// TIA Portal V17 export
// export: Created 2025-03-05T08:02:40.8398628Z, ExportSetting WithDefaults, DisplayName Totally Integrated Automation Portal, DisplayVersion V17 Update 8, DisplayName TIA Portal Openness, DisplayVersion V17 Update 8, DisplayName TIA Portal Version Control Interface, DisplayVersion V17, DisplayName SINAMICS Startdrive Advanced, DisplayVersion V17 SP2, DisplayName SINAMICS Startdrive G110M, G120, G120C, G120D, G120P, G115D, DisplayVersion V17 SP2, DisplayName SINAMICS Startdrive G130, G150, S120, S150, SINAMICS MV, S210, DisplayVersion V17 SP2, DisplayName STEP 7 Professional, DisplayVersion V17 Update 8, DisplayName SINUMERIK ONE STEP 7 Toolbox, DisplayVersion V17 Update 12, DisplayName SINUMERIK 840D sl STEP 7 Toolbox, DisplayVersion V17 Update 12, DisplayName STEP 7 Safety, DisplayVersion V17 Update 6, DisplayName WinCC Advanced, DisplayVersion V17 Update 8
FUNCTION "FC441_POWDER_FEEDERS_ALARM_DECODING" : Void   // FC441, LAD
{ S7_Optimized_Access := 'FALSE' }
AUTHOR : ETXETAR
VERSION : 1.0
// stored: AutoNumber false, IsIECCheckEnabled false, SetENOAutomatically false, UDAEnableTagReadback false
   VAR_TEMP
      RST_ALARMS_1 : Bool;   // RESET ALARMS 1
      RST_ALARMS_2 : Bool;   // RESET ALARMS 2
      ZERO : Int;   // ZERO
      RET_VAL_1 : Int;   // RET VALUE
   END_VAR
   VAR CONSTANT
      FC_CONSTANT : Int := 442;
   END_VAR
   VAR_TEMP   // added for the SCL form of the ladder/FBD networks
      _w1 : Bool;
      _w2 : Bool;
      _w3 : Bool;
   END_VAR
BEGIN

REGION Network 1: ZERO
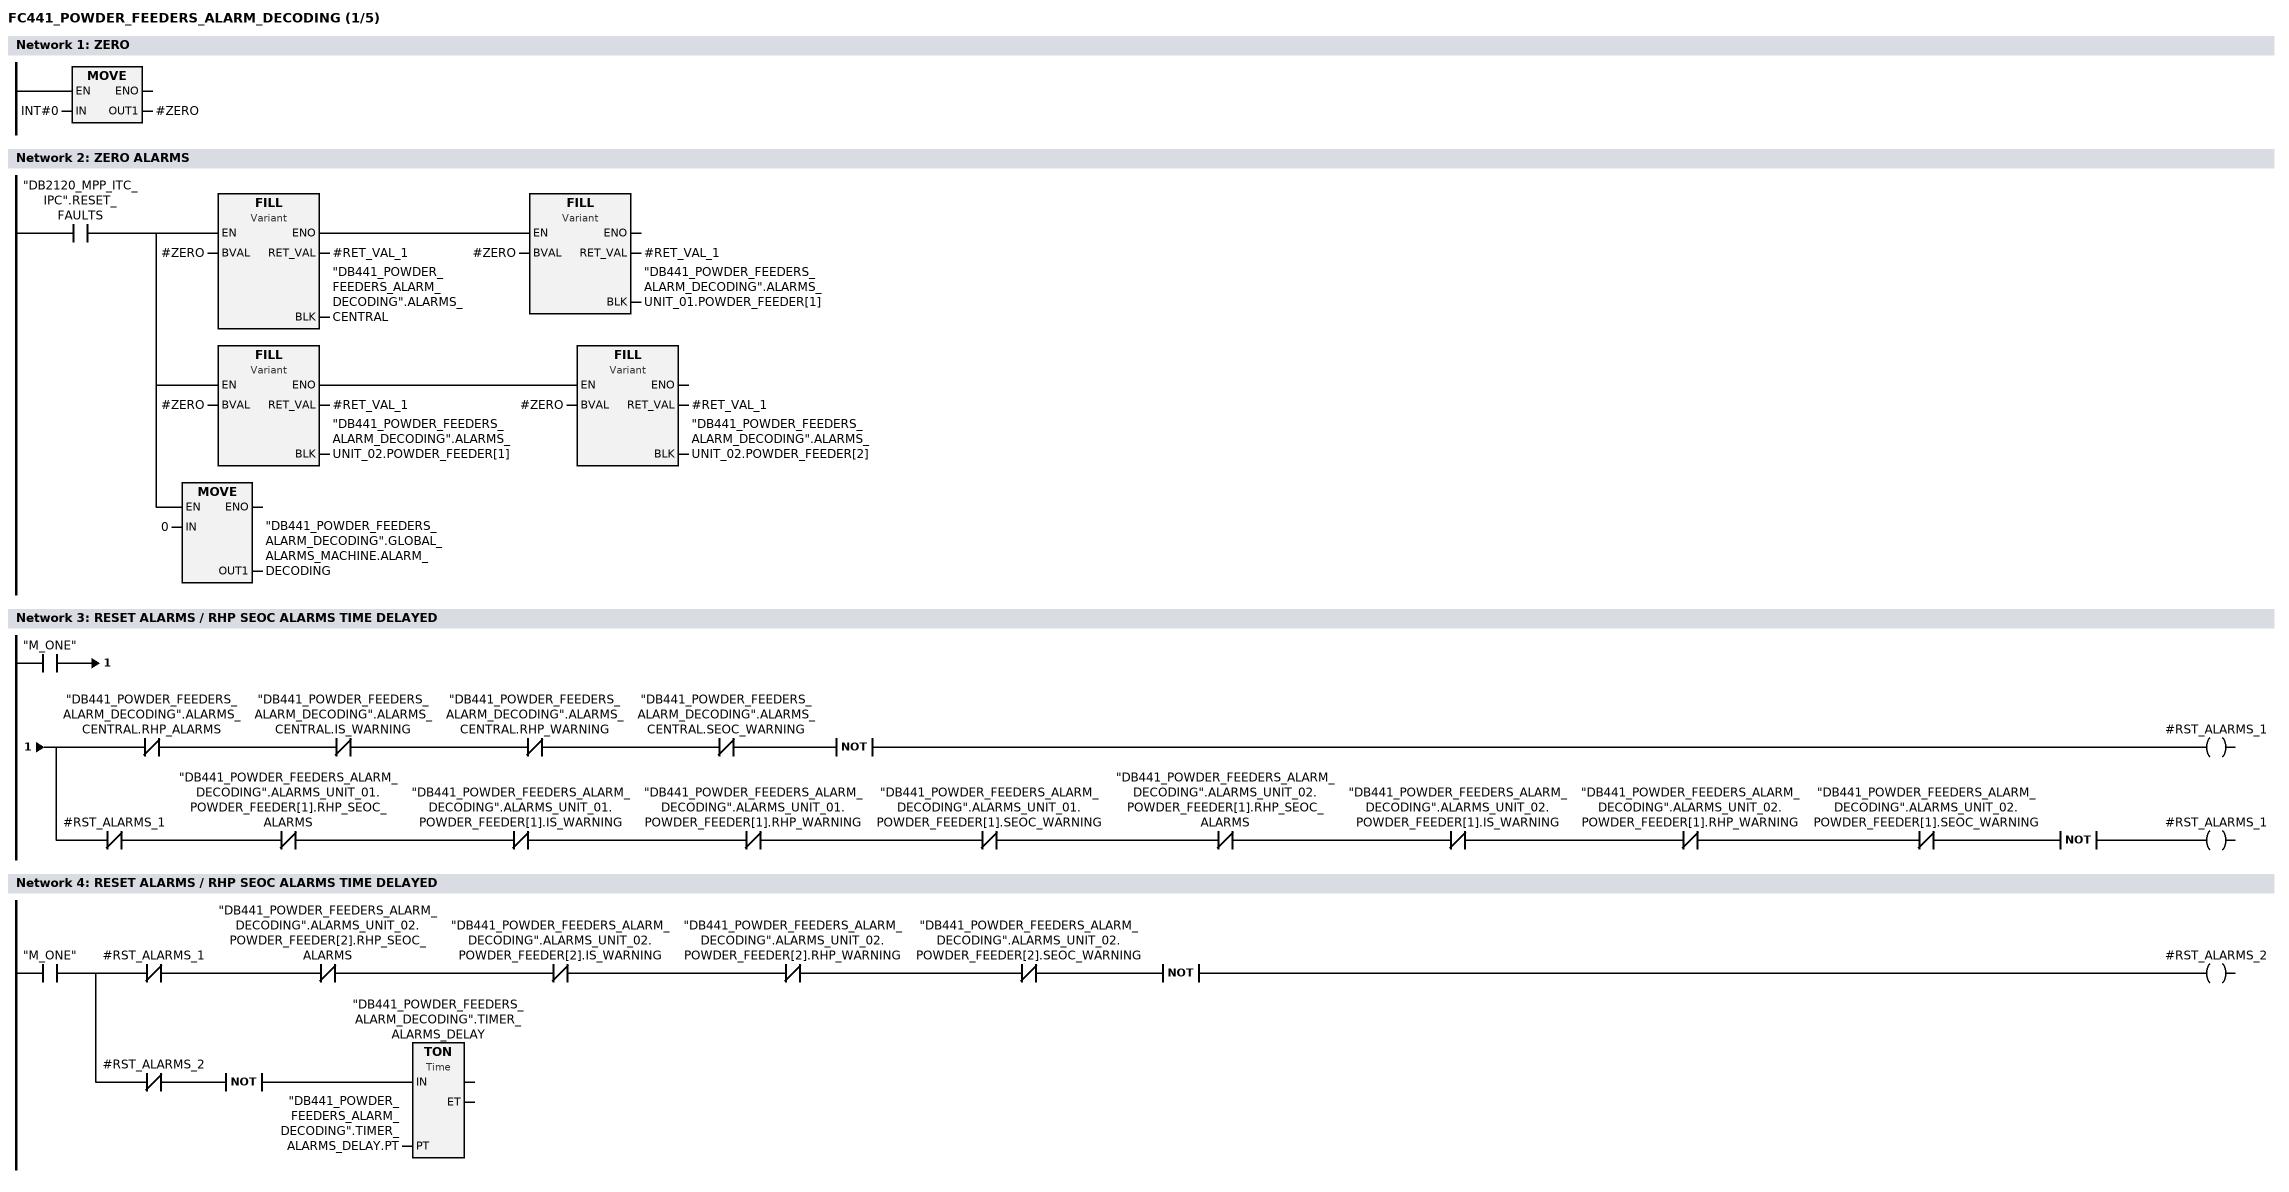
   RUNG wire#powerrail
      { S7_GenerateENO := "TRUE" } Move(in := INT#0, out1 => #ZERO)
   END_RUNG
   // the same network as SCL:
   #ZERO := INT#0;
END_REGION

REGION Network 2: ZERO ALARMS
   RUNG wire#powerrail
      Contact( "DB2120_MPP_ITC_IPC".RESET_FAULTS )
      wire#w1
      { S7_Templates := "ptr_type := Variant" } FILL(BVAL := #ZERO, RET_VAL => #RET_VAL_1, BLK => "DB441_POWDER_FEEDERS_ALARM_DECODING".ALARMS_CENTRAL)
      { S7_Templates := "ptr_type := Variant" } FILL(BVAL := #ZERO, RET_VAL => #RET_VAL_1, BLK => "DB441_POWDER_FEEDERS_ALARM_DECODING".ALARMS_UNIT_01.POWDER_FEEDER[1])
   END_RUNG
   RUNG wire#w1
      { S7_Templates := "ptr_type := Variant" } FILL(BVAL := #ZERO, RET_VAL => #RET_VAL_1, BLK => "DB441_POWDER_FEEDERS_ALARM_DECODING".ALARMS_UNIT_02.POWDER_FEEDER[1])
      { S7_Templates := "ptr_type := Variant" } FILL(BVAL := #ZERO, RET_VAL => #RET_VAL_1, BLK => "DB441_POWDER_FEEDERS_ALARM_DECODING".ALARMS_UNIT_02.POWDER_FEEDER[2])
   END_RUNG
   RUNG wire#w1
      { S7_GenerateENO := "TRUE" } Move(in := 0, out1 => "DB441_POWDER_FEEDERS_ALARM_DECODING".GLOBAL_ALARMS_MACHINE.ALARM_DECODING)
   END_RUNG
   // the same network as SCL:
   #_w2 := "DB2120_MPP_ITC_IPC".RESET_FAULTS;
   #RET_VAL_1 := FILL(EN := "DB2120_MPP_ITC_IPC".RESET_FAULTS,
                      BVAL := #ZERO,
                      BLK => "DB441_POWDER_FEEDERS_ALARM_DECODING".ALARMS_CENTRAL,
                      ENO => #_w1);
   IF #_w1 THEN
       #RET_VAL_1 := FILL(BVAL := #ZERO,
                          BLK => "DB441_POWDER_FEEDERS_ALARM_DECODING".ALARMS_UNIT_01.POWDER_FEEDER[1]);
   END_IF;
   #RET_VAL_1 := FILL(EN := #_w2,
                      BVAL := #ZERO,
                      BLK => "DB441_POWDER_FEEDERS_ALARM_DECODING".ALARMS_UNIT_02.POWDER_FEEDER[1],
                      ENO => #_w3);
   IF #_w3 THEN
       #RET_VAL_1 := FILL(BVAL := #ZERO,
                          BLK => "DB441_POWDER_FEEDERS_ALARM_DECODING".ALARMS_UNIT_02.POWDER_FEEDER[2]);
   END_IF;
   IF #_w2 THEN "DB441_POWDER_FEEDERS_ALARM_DECODING".GLOBAL_ALARMS_MACHINE.ALARM_DECODING := 0; END_IF;
END_REGION

REGION Network 3: RESET ALARMS / RHP SEOC ALARMS TIME DELAYED
   RUNG wire#powerrail
      Contact( "M_ONE" )
      wire#w1
      I_Contact( "DB441_POWDER_FEEDERS_ALARM_DECODING".ALARMS_CENTRAL.RHP_ALARMS )
      I_Contact( "DB441_POWDER_FEEDERS_ALARM_DECODING".ALARMS_CENTRAL.IS_WARNING )
      I_Contact( "DB441_POWDER_FEEDERS_ALARM_DECODING".ALARMS_CENTRAL.RHP_WARNING )
      I_Contact( "DB441_POWDER_FEEDERS_ALARM_DECODING".ALARMS_CENTRAL.SEOC_WARNING )
      Not()
      Coil( #RST_ALARMS_1 )
   END_RUNG
   RUNG wire#w1
      I_Contact( #RST_ALARMS_1 )
      I_Contact( "DB441_POWDER_FEEDERS_ALARM_DECODING".ALARMS_UNIT_01.POWDER_FEEDER[1].RHP_SEOC_ALARMS )
      I_Contact( "DB441_POWDER_FEEDERS_ALARM_DECODING".ALARMS_UNIT_01.POWDER_FEEDER[1].IS_WARNING )
      I_Contact( "DB441_POWDER_FEEDERS_ALARM_DECODING".ALARMS_UNIT_01.POWDER_FEEDER[1].RHP_WARNING )
      I_Contact( "DB441_POWDER_FEEDERS_ALARM_DECODING".ALARMS_UNIT_01.POWDER_FEEDER[1].SEOC_WARNING )
      I_Contact( "DB441_POWDER_FEEDERS_ALARM_DECODING".ALARMS_UNIT_02.POWDER_FEEDER[1].RHP_SEOC_ALARMS )
      I_Contact( "DB441_POWDER_FEEDERS_ALARM_DECODING".ALARMS_UNIT_02.POWDER_FEEDER[1].IS_WARNING )
      I_Contact( "DB441_POWDER_FEEDERS_ALARM_DECODING".ALARMS_UNIT_02.POWDER_FEEDER[1].RHP_WARNING )
      I_Contact( "DB441_POWDER_FEEDERS_ALARM_DECODING".ALARMS_UNIT_02.POWDER_FEEDER[1].SEOC_WARNING )
      Not()
      Coil( #RST_ALARMS_1 )
   END_RUNG
   // the same network as SCL:
   #RST_ALARMS_1 := NOT ("M_ONE" AND NOT "DB441_POWDER_FEEDERS_ALARM_DECODING".ALARMS_CENTRAL.RHP_ALARMS AND NOT "DB441_POWDER_FEEDERS_ALARM_DECODING".ALARMS_CENTRAL.IS_WARNING AND NOT "DB441_POWDER_FEEDERS_ALARM_DECODING".ALARMS_CENTRAL.RHP_WARNING AND NOT "DB441_POWDER_FEEDERS_ALARM_DECODING".ALARMS_CENTRAL.SEOC_WARNING);
   #RST_ALARMS_1 := NOT ("M_ONE" AND NOT #RST_ALARMS_1 AND NOT "DB441_POWDER_FEEDERS_ALARM_DECODING".ALARMS_UNIT_01.POWDER_FEEDER[1].RHP_SEOC_ALARMS AND NOT "DB441_POWDER_FEEDERS_ALARM_DECODING".ALARMS_UNIT_01.POWDER_FEEDER[1].IS_WARNING AND NOT "DB441_POWDER_FEEDERS_ALARM_DECODING".ALARMS_UNIT_01.POWDER_FEEDER[1].RHP_WARNING AND NOT "DB441_POWDER_FEEDERS_ALARM_DECODING".ALARMS_UNIT_01.POWDER_FEEDER[1].SEOC_WARNING AND NOT "DB441_POWDER_FEEDERS_ALARM_DECODING".ALARMS_UNIT_02.POWDER_FEEDER[1].RHP_SEOC_ALARMS AND NOT "DB441_POWDER_FEEDERS_ALARM_DECODING".ALARMS_UNIT_02.POWDER_FEEDER[1].IS_WARNING AND NOT "DB441_POWDER_FEEDERS_ALARM_DECODING".ALARMS_UNIT_02.POWDER_FEEDER[1].RHP_WARNING AND NOT "DB441_POWDER_FEEDERS_ALARM_DECODING".ALARMS_UNIT_02.POWDER_FEEDER[1].SEOC_WARNING);
END_REGION

REGION Network 4: RESET ALARMS / RHP SEOC ALARMS TIME DELAYED
   RUNG wire#powerrail
      Contact( "M_ONE" )
      wire#w1
      I_Contact( #RST_ALARMS_1 )
      I_Contact( "DB441_POWDER_FEEDERS_ALARM_DECODING".ALARMS_UNIT_02.POWDER_FEEDER[2].RHP_SEOC_ALARMS )
      I_Contact( "DB441_POWDER_FEEDERS_ALARM_DECODING".ALARMS_UNIT_02.POWDER_FEEDER[2].IS_WARNING )
      I_Contact( "DB441_POWDER_FEEDERS_ALARM_DECODING".ALARMS_UNIT_02.POWDER_FEEDER[2].RHP_WARNING )
      I_Contact( "DB441_POWDER_FEEDERS_ALARM_DECODING".ALARMS_UNIT_02.POWDER_FEEDER[2].SEOC_WARNING )
      Not()
      Coil( #RST_ALARMS_2 )
   END_RUNG
   RUNG wire#w1
      I_Contact( #RST_ALARMS_2 )
      Not()
      { S7_Templates := "time_type := Time" } "DB441_POWDER_FEEDERS_ALARM_DECODING".TIMER_ALARMS_DELAY.TON(pt := "DB441_POWDER_FEEDERS_ALARM_DECODING".TIMER_ALARMS_DELAY.PT, et =>)
   END_RUNG
   // the same network as SCL:
   #RST_ALARMS_2 := NOT ("M_ONE" AND NOT #RST_ALARMS_1 AND NOT "DB441_POWDER_FEEDERS_ALARM_DECODING".ALARMS_UNIT_02.POWDER_FEEDER[2].RHP_SEOC_ALARMS AND NOT "DB441_POWDER_FEEDERS_ALARM_DECODING".ALARMS_UNIT_02.POWDER_FEEDER[2].IS_WARNING AND NOT "DB441_POWDER_FEEDERS_ALARM_DECODING".ALARMS_UNIT_02.POWDER_FEEDER[2].RHP_WARNING AND NOT "DB441_POWDER_FEEDERS_ALARM_DECODING".ALARMS_UNIT_02.POWDER_FEEDER[2].SEOC_WARNING);
   "DB441_POWDER_FEEDERS_ALARM_DECODING".TIMER_ALARMS_DELAY.TON(IN := NOT ("M_ONE" AND NOT #RST_ALARMS_2),
                           PT := "DB441_POWDER_FEEDERS_ALARM_DECODING".TIMER_ALARMS_DELAY.PT);
END_REGION

REGION Network 5: CENTRAL ALARMS AND UNIT 01 FEEDERS ALARMS RESET / RETURN HOME POSITION & STOP END OF CYCLE ALARMS
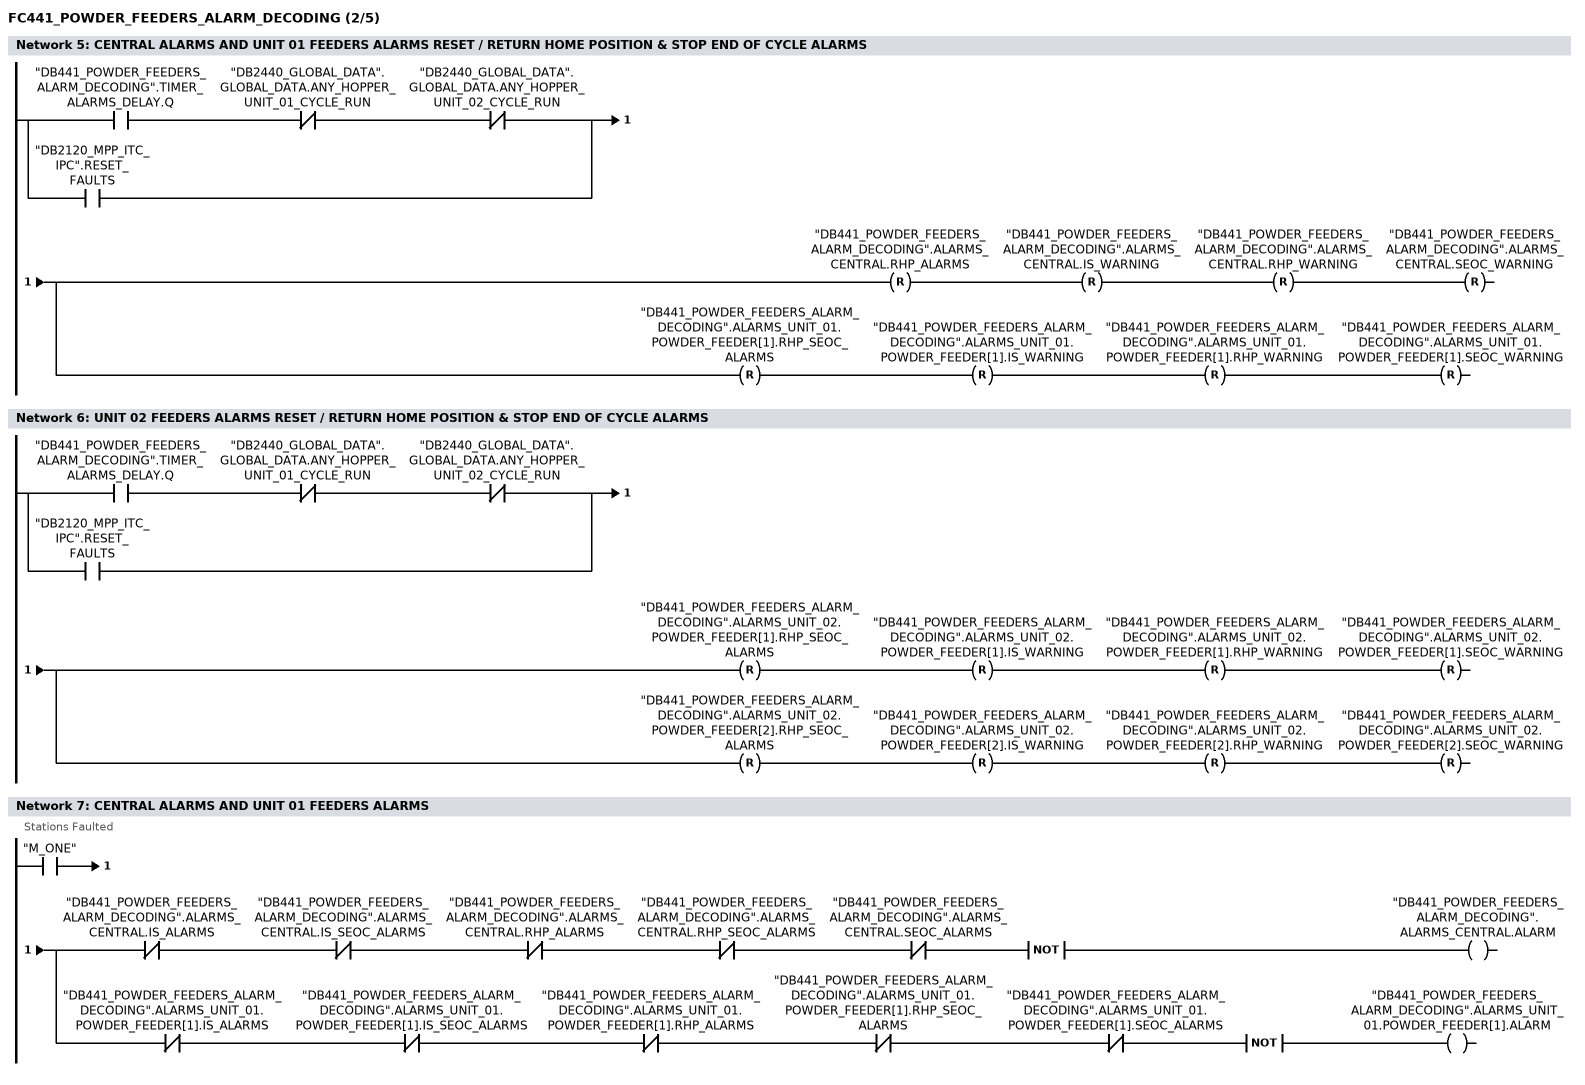
   RUNG wire#powerrail
      Contact( "DB441_POWDER_FEEDERS_ALARM_DECODING".TIMER_ALARMS_DELAY.Q )
      I_Contact( "DB2440_GLOBAL_DATA".GLOBAL_DATA.ANY_HOPPER_UNIT_01_CYCLE_RUN )
      I_Contact( "DB2440_GLOBAL_DATA".GLOBAL_DATA.ANY_HOPPER_UNIT_02_CYCLE_RUN )
      wire#w1
      R_Coil( "DB441_POWDER_FEEDERS_ALARM_DECODING".ALARMS_CENTRAL.RHP_ALARMS )
      R_Coil( "DB441_POWDER_FEEDERS_ALARM_DECODING".ALARMS_CENTRAL.IS_WARNING )
      R_Coil( "DB441_POWDER_FEEDERS_ALARM_DECODING".ALARMS_CENTRAL.RHP_WARNING )
      R_Coil( "DB441_POWDER_FEEDERS_ALARM_DECODING".ALARMS_CENTRAL.SEOC_WARNING )
   END_RUNG
   RUNG wire#powerrail
      Contact( "DB2120_MPP_ITC_IPC".RESET_FAULTS )
   END_RUNG wire#w1
   RUNG wire#w1
      R_Coil( "DB441_POWDER_FEEDERS_ALARM_DECODING".ALARMS_UNIT_01.POWDER_FEEDER[1].RHP_SEOC_ALARMS )
      R_Coil( "DB441_POWDER_FEEDERS_ALARM_DECODING".ALARMS_UNIT_01.POWDER_FEEDER[1].IS_WARNING )
      R_Coil( "DB441_POWDER_FEEDERS_ALARM_DECODING".ALARMS_UNIT_01.POWDER_FEEDER[1].RHP_WARNING )
      R_Coil( "DB441_POWDER_FEEDERS_ALARM_DECODING".ALARMS_UNIT_01.POWDER_FEEDER[1].SEOC_WARNING )
   END_RUNG
   // the same network as SCL:
   IF ("DB441_POWDER_FEEDERS_ALARM_DECODING".TIMER_ALARMS_DELAY.Q AND NOT "DB2440_GLOBAL_DATA".GLOBAL_DATA.ANY_HOPPER_UNIT_01_CYCLE_RUN AND NOT "DB2440_GLOBAL_DATA".GLOBAL_DATA.ANY_HOPPER_UNIT_02_CYCLE_RUN) OR "DB2120_MPP_ITC_IPC".RESET_FAULTS THEN
       "DB441_POWDER_FEEDERS_ALARM_DECODING".ALARMS_CENTRAL.RHP_ALARMS := FALSE;
       "DB441_POWDER_FEEDERS_ALARM_DECODING".ALARMS_CENTRAL.IS_WARNING := FALSE;
       "DB441_POWDER_FEEDERS_ALARM_DECODING".ALARMS_CENTRAL.RHP_WARNING := FALSE;
       "DB441_POWDER_FEEDERS_ALARM_DECODING".ALARMS_CENTRAL.SEOC_WARNING := FALSE;
       "DB441_POWDER_FEEDERS_ALARM_DECODING".ALARMS_UNIT_01.POWDER_FEEDER[1].RHP_SEOC_ALARMS := FALSE;
       "DB441_POWDER_FEEDERS_ALARM_DECODING".ALARMS_UNIT_01.POWDER_FEEDER[1].IS_WARNING := FALSE;
       "DB441_POWDER_FEEDERS_ALARM_DECODING".ALARMS_UNIT_01.POWDER_FEEDER[1].RHP_WARNING := FALSE;
       "DB441_POWDER_FEEDERS_ALARM_DECODING".ALARMS_UNIT_01.POWDER_FEEDER[1].SEOC_WARNING := FALSE;
   END_IF;
END_REGION

REGION Network 6: UNIT 02 FEEDERS ALARMS RESET / RETURN HOME POSITION & STOP END OF CYCLE ALARMS
   RUNG wire#powerrail
      Contact( "DB441_POWDER_FEEDERS_ALARM_DECODING".TIMER_ALARMS_DELAY.Q )
      I_Contact( "DB2440_GLOBAL_DATA".GLOBAL_DATA.ANY_HOPPER_UNIT_01_CYCLE_RUN )
      I_Contact( "DB2440_GLOBAL_DATA".GLOBAL_DATA.ANY_HOPPER_UNIT_02_CYCLE_RUN )
      wire#w1
      R_Coil( "DB441_POWDER_FEEDERS_ALARM_DECODING".ALARMS_UNIT_02.POWDER_FEEDER[1].RHP_SEOC_ALARMS )
      R_Coil( "DB441_POWDER_FEEDERS_ALARM_DECODING".ALARMS_UNIT_02.POWDER_FEEDER[1].IS_WARNING )
      R_Coil( "DB441_POWDER_FEEDERS_ALARM_DECODING".ALARMS_UNIT_02.POWDER_FEEDER[1].RHP_WARNING )
      R_Coil( "DB441_POWDER_FEEDERS_ALARM_DECODING".ALARMS_UNIT_02.POWDER_FEEDER[1].SEOC_WARNING )
   END_RUNG
   RUNG wire#powerrail
      Contact( "DB2120_MPP_ITC_IPC".RESET_FAULTS )
   END_RUNG wire#w1
   RUNG wire#w1
      R_Coil( "DB441_POWDER_FEEDERS_ALARM_DECODING".ALARMS_UNIT_02.POWDER_FEEDER[2].RHP_SEOC_ALARMS )
      R_Coil( "DB441_POWDER_FEEDERS_ALARM_DECODING".ALARMS_UNIT_02.POWDER_FEEDER[2].IS_WARNING )
      R_Coil( "DB441_POWDER_FEEDERS_ALARM_DECODING".ALARMS_UNIT_02.POWDER_FEEDER[2].RHP_WARNING )
      R_Coil( "DB441_POWDER_FEEDERS_ALARM_DECODING".ALARMS_UNIT_02.POWDER_FEEDER[2].SEOC_WARNING )
   END_RUNG
   // the same network as SCL:
   IF ("DB441_POWDER_FEEDERS_ALARM_DECODING".TIMER_ALARMS_DELAY.Q AND NOT "DB2440_GLOBAL_DATA".GLOBAL_DATA.ANY_HOPPER_UNIT_01_CYCLE_RUN AND NOT "DB2440_GLOBAL_DATA".GLOBAL_DATA.ANY_HOPPER_UNIT_02_CYCLE_RUN) OR "DB2120_MPP_ITC_IPC".RESET_FAULTS THEN
       "DB441_POWDER_FEEDERS_ALARM_DECODING".ALARMS_UNIT_02.POWDER_FEEDER[1].RHP_SEOC_ALARMS := FALSE;
       "DB441_POWDER_FEEDERS_ALARM_DECODING".ALARMS_UNIT_02.POWDER_FEEDER[1].IS_WARNING := FALSE;
       "DB441_POWDER_FEEDERS_ALARM_DECODING".ALARMS_UNIT_02.POWDER_FEEDER[1].RHP_WARNING := FALSE;
       "DB441_POWDER_FEEDERS_ALARM_DECODING".ALARMS_UNIT_02.POWDER_FEEDER[1].SEOC_WARNING := FALSE;
       "DB441_POWDER_FEEDERS_ALARM_DECODING".ALARMS_UNIT_02.POWDER_FEEDER[2].RHP_SEOC_ALARMS := FALSE;
       "DB441_POWDER_FEEDERS_ALARM_DECODING".ALARMS_UNIT_02.POWDER_FEEDER[2].IS_WARNING := FALSE;
       "DB441_POWDER_FEEDERS_ALARM_DECODING".ALARMS_UNIT_02.POWDER_FEEDER[2].RHP_WARNING := FALSE;
       "DB441_POWDER_FEEDERS_ALARM_DECODING".ALARMS_UNIT_02.POWDER_FEEDER[2].SEOC_WARNING := FALSE;
   END_IF;
END_REGION

REGION Network 7: CENTRAL ALARMS AND UNIT 01 FEEDERS ALARMS
   // Stations Faulted
   RUNG wire#powerrail
      Contact( "M_ONE" )
      wire#w1
      I_Contact( "DB441_POWDER_FEEDERS_ALARM_DECODING".ALARMS_CENTRAL.IS_ALARMS )
      I_Contact( "DB441_POWDER_FEEDERS_ALARM_DECODING".ALARMS_CENTRAL.IS_SEOC_ALARMS )
      I_Contact( "DB441_POWDER_FEEDERS_ALARM_DECODING".ALARMS_CENTRAL.RHP_ALARMS )
      I_Contact( "DB441_POWDER_FEEDERS_ALARM_DECODING".ALARMS_CENTRAL.RHP_SEOC_ALARMS )
      I_Contact( "DB441_POWDER_FEEDERS_ALARM_DECODING".ALARMS_CENTRAL.SEOC_ALARMS )
      Not()
      Coil( "DB441_POWDER_FEEDERS_ALARM_DECODING".ALARMS_CENTRAL.ALARM )
   END_RUNG
   RUNG wire#w1
      I_Contact( "DB441_POWDER_FEEDERS_ALARM_DECODING".ALARMS_UNIT_01.POWDER_FEEDER[1].IS_ALARMS )
      I_Contact( "DB441_POWDER_FEEDERS_ALARM_DECODING".ALARMS_UNIT_01.POWDER_FEEDER[1].IS_SEOC_ALARMS )
      I_Contact( "DB441_POWDER_FEEDERS_ALARM_DECODING".ALARMS_UNIT_01.POWDER_FEEDER[1].RHP_ALARMS )
      I_Contact( "DB441_POWDER_FEEDERS_ALARM_DECODING".ALARMS_UNIT_01.POWDER_FEEDER[1].RHP_SEOC_ALARMS )
      I_Contact( "DB441_POWDER_FEEDERS_ALARM_DECODING".ALARMS_UNIT_01.POWDER_FEEDER[1].SEOC_ALARMS )
      Not()
      Coil( "DB441_POWDER_FEEDERS_ALARM_DECODING".ALARMS_UNIT_01.POWDER_FEEDER[1].ALARM )
   END_RUNG
   // the same network as SCL:
   "DB441_POWDER_FEEDERS_ALARM_DECODING".ALARMS_CENTRAL.ALARM := NOT ("M_ONE" AND NOT "DB441_POWDER_FEEDERS_ALARM_DECODING".ALARMS_CENTRAL.IS_ALARMS AND NOT "DB441_POWDER_FEEDERS_ALARM_DECODING".ALARMS_CENTRAL.IS_SEOC_ALARMS AND NOT "DB441_POWDER_FEEDERS_ALARM_DECODING".ALARMS_CENTRAL.RHP_ALARMS AND NOT "DB441_POWDER_FEEDERS_ALARM_DECODING".ALARMS_CENTRAL.RHP_SEOC_ALARMS AND NOT "DB441_POWDER_FEEDERS_ALARM_DECODING".ALARMS_CENTRAL.SEOC_ALARMS);
   "DB441_POWDER_FEEDERS_ALARM_DECODING".ALARMS_UNIT_01.POWDER_FEEDER[1].ALARM := NOT ("M_ONE" AND NOT "DB441_POWDER_FEEDERS_ALARM_DECODING".ALARMS_UNIT_01.POWDER_FEEDER[1].IS_ALARMS AND NOT "DB441_POWDER_FEEDERS_ALARM_DECODING".ALARMS_UNIT_01.POWDER_FEEDER[1].IS_SEOC_ALARMS AND NOT "DB441_POWDER_FEEDERS_ALARM_DECODING".ALARMS_UNIT_01.POWDER_FEEDER[1].RHP_ALARMS AND NOT "DB441_POWDER_FEEDERS_ALARM_DECODING".ALARMS_UNIT_01.POWDER_FEEDER[1].RHP_SEOC_ALARMS AND NOT "DB441_POWDER_FEEDERS_ALARM_DECODING".ALARMS_UNIT_01.POWDER_FEEDER[1].SEOC_ALARMS);
END_REGION

REGION Network 8: UNIT 02 FEEDERS ALARMS
   // Stations Faulted
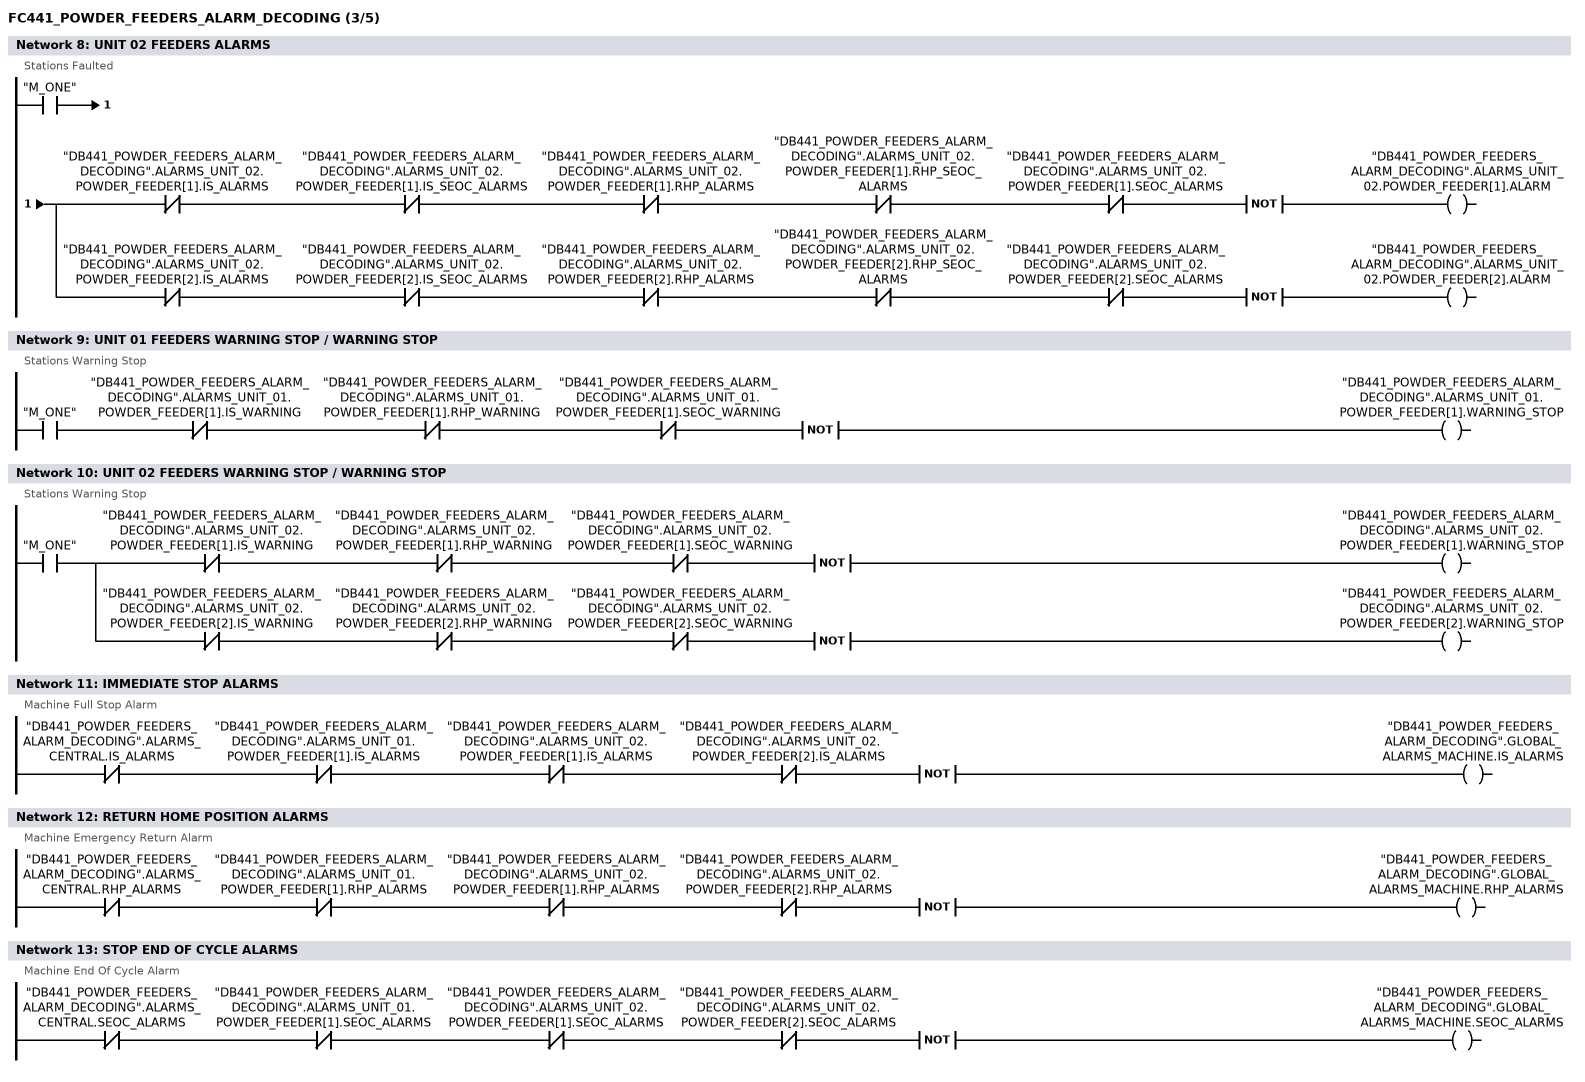
   RUNG wire#powerrail
      Contact( "M_ONE" )
      wire#w1
      I_Contact( "DB441_POWDER_FEEDERS_ALARM_DECODING".ALARMS_UNIT_02.POWDER_FEEDER[1].IS_ALARMS )
      I_Contact( "DB441_POWDER_FEEDERS_ALARM_DECODING".ALARMS_UNIT_02.POWDER_FEEDER[1].IS_SEOC_ALARMS )
      I_Contact( "DB441_POWDER_FEEDERS_ALARM_DECODING".ALARMS_UNIT_02.POWDER_FEEDER[1].RHP_ALARMS )
      I_Contact( "DB441_POWDER_FEEDERS_ALARM_DECODING".ALARMS_UNIT_02.POWDER_FEEDER[1].RHP_SEOC_ALARMS )
      I_Contact( "DB441_POWDER_FEEDERS_ALARM_DECODING".ALARMS_UNIT_02.POWDER_FEEDER[1].SEOC_ALARMS )
      Not()
      Coil( "DB441_POWDER_FEEDERS_ALARM_DECODING".ALARMS_UNIT_02.POWDER_FEEDER[1].ALARM )
   END_RUNG
   RUNG wire#w1
      I_Contact( "DB441_POWDER_FEEDERS_ALARM_DECODING".ALARMS_UNIT_02.POWDER_FEEDER[2].IS_ALARMS )
      I_Contact( "DB441_POWDER_FEEDERS_ALARM_DECODING".ALARMS_UNIT_02.POWDER_FEEDER[2].IS_SEOC_ALARMS )
      I_Contact( "DB441_POWDER_FEEDERS_ALARM_DECODING".ALARMS_UNIT_02.POWDER_FEEDER[2].RHP_ALARMS )
      I_Contact( "DB441_POWDER_FEEDERS_ALARM_DECODING".ALARMS_UNIT_02.POWDER_FEEDER[2].RHP_SEOC_ALARMS )
      I_Contact( "DB441_POWDER_FEEDERS_ALARM_DECODING".ALARMS_UNIT_02.POWDER_FEEDER[2].SEOC_ALARMS )
      Not()
      Coil( "DB441_POWDER_FEEDERS_ALARM_DECODING".ALARMS_UNIT_02.POWDER_FEEDER[2].ALARM )
   END_RUNG
   // the same network as SCL:
   "DB441_POWDER_FEEDERS_ALARM_DECODING".ALARMS_UNIT_02.POWDER_FEEDER[1].ALARM := NOT ("M_ONE" AND NOT "DB441_POWDER_FEEDERS_ALARM_DECODING".ALARMS_UNIT_02.POWDER_FEEDER[1].IS_ALARMS AND NOT "DB441_POWDER_FEEDERS_ALARM_DECODING".ALARMS_UNIT_02.POWDER_FEEDER[1].IS_SEOC_ALARMS AND NOT "DB441_POWDER_FEEDERS_ALARM_DECODING".ALARMS_UNIT_02.POWDER_FEEDER[1].RHP_ALARMS AND NOT "DB441_POWDER_FEEDERS_ALARM_DECODING".ALARMS_UNIT_02.POWDER_FEEDER[1].RHP_SEOC_ALARMS AND NOT "DB441_POWDER_FEEDERS_ALARM_DECODING".ALARMS_UNIT_02.POWDER_FEEDER[1].SEOC_ALARMS);
   "DB441_POWDER_FEEDERS_ALARM_DECODING".ALARMS_UNIT_02.POWDER_FEEDER[2].ALARM := NOT ("M_ONE" AND NOT "DB441_POWDER_FEEDERS_ALARM_DECODING".ALARMS_UNIT_02.POWDER_FEEDER[2].IS_ALARMS AND NOT "DB441_POWDER_FEEDERS_ALARM_DECODING".ALARMS_UNIT_02.POWDER_FEEDER[2].IS_SEOC_ALARMS AND NOT "DB441_POWDER_FEEDERS_ALARM_DECODING".ALARMS_UNIT_02.POWDER_FEEDER[2].RHP_ALARMS AND NOT "DB441_POWDER_FEEDERS_ALARM_DECODING".ALARMS_UNIT_02.POWDER_FEEDER[2].RHP_SEOC_ALARMS AND NOT "DB441_POWDER_FEEDERS_ALARM_DECODING".ALARMS_UNIT_02.POWDER_FEEDER[2].SEOC_ALARMS);
END_REGION

REGION Network 9: UNIT 01 FEEDERS WARNING STOP / WARNING STOP
   // Stations Warning Stop
   RUNG wire#powerrail
      Contact( "M_ONE" )
      I_Contact( "DB441_POWDER_FEEDERS_ALARM_DECODING".ALARMS_UNIT_01.POWDER_FEEDER[1].IS_WARNING )
      I_Contact( "DB441_POWDER_FEEDERS_ALARM_DECODING".ALARMS_UNIT_01.POWDER_FEEDER[1].RHP_WARNING )
      I_Contact( "DB441_POWDER_FEEDERS_ALARM_DECODING".ALARMS_UNIT_01.POWDER_FEEDER[1].SEOC_WARNING )
      Not()
      Coil( "DB441_POWDER_FEEDERS_ALARM_DECODING".ALARMS_UNIT_01.POWDER_FEEDER[1].WARNING_STOP )
   END_RUNG
   // the same network as SCL:
   "DB441_POWDER_FEEDERS_ALARM_DECODING".ALARMS_UNIT_01.POWDER_FEEDER[1].WARNING_STOP := NOT ("M_ONE" AND NOT "DB441_POWDER_FEEDERS_ALARM_DECODING".ALARMS_UNIT_01.POWDER_FEEDER[1].IS_WARNING AND NOT "DB441_POWDER_FEEDERS_ALARM_DECODING".ALARMS_UNIT_01.POWDER_FEEDER[1].RHP_WARNING AND NOT "DB441_POWDER_FEEDERS_ALARM_DECODING".ALARMS_UNIT_01.POWDER_FEEDER[1].SEOC_WARNING);
END_REGION

REGION Network 10: UNIT 02 FEEDERS WARNING STOP / WARNING STOP
   // Stations Warning Stop
   RUNG wire#powerrail
      Contact( "M_ONE" )
      wire#w1
      I_Contact( "DB441_POWDER_FEEDERS_ALARM_DECODING".ALARMS_UNIT_02.POWDER_FEEDER[1].IS_WARNING )
      I_Contact( "DB441_POWDER_FEEDERS_ALARM_DECODING".ALARMS_UNIT_02.POWDER_FEEDER[1].RHP_WARNING )
      I_Contact( "DB441_POWDER_FEEDERS_ALARM_DECODING".ALARMS_UNIT_02.POWDER_FEEDER[1].SEOC_WARNING )
      Not()
      Coil( "DB441_POWDER_FEEDERS_ALARM_DECODING".ALARMS_UNIT_02.POWDER_FEEDER[1].WARNING_STOP )
   END_RUNG
   RUNG wire#w1
      I_Contact( "DB441_POWDER_FEEDERS_ALARM_DECODING".ALARMS_UNIT_02.POWDER_FEEDER[2].IS_WARNING )
      I_Contact( "DB441_POWDER_FEEDERS_ALARM_DECODING".ALARMS_UNIT_02.POWDER_FEEDER[2].RHP_WARNING )
      I_Contact( "DB441_POWDER_FEEDERS_ALARM_DECODING".ALARMS_UNIT_02.POWDER_FEEDER[2].SEOC_WARNING )
      Not()
      Coil( "DB441_POWDER_FEEDERS_ALARM_DECODING".ALARMS_UNIT_02.POWDER_FEEDER[2].WARNING_STOP )
   END_RUNG
   // the same network as SCL:
   "DB441_POWDER_FEEDERS_ALARM_DECODING".ALARMS_UNIT_02.POWDER_FEEDER[1].WARNING_STOP := NOT ("M_ONE" AND NOT "DB441_POWDER_FEEDERS_ALARM_DECODING".ALARMS_UNIT_02.POWDER_FEEDER[1].IS_WARNING AND NOT "DB441_POWDER_FEEDERS_ALARM_DECODING".ALARMS_UNIT_02.POWDER_FEEDER[1].RHP_WARNING AND NOT "DB441_POWDER_FEEDERS_ALARM_DECODING".ALARMS_UNIT_02.POWDER_FEEDER[1].SEOC_WARNING);
   "DB441_POWDER_FEEDERS_ALARM_DECODING".ALARMS_UNIT_02.POWDER_FEEDER[2].WARNING_STOP := NOT ("M_ONE" AND NOT "DB441_POWDER_FEEDERS_ALARM_DECODING".ALARMS_UNIT_02.POWDER_FEEDER[2].IS_WARNING AND NOT "DB441_POWDER_FEEDERS_ALARM_DECODING".ALARMS_UNIT_02.POWDER_FEEDER[2].RHP_WARNING AND NOT "DB441_POWDER_FEEDERS_ALARM_DECODING".ALARMS_UNIT_02.POWDER_FEEDER[2].SEOC_WARNING);
END_REGION

REGION Network 11: IMMEDIATE STOP ALARMS
   // Machine Full Stop Alarm
   RUNG wire#powerrail
      I_Contact( "DB441_POWDER_FEEDERS_ALARM_DECODING".ALARMS_CENTRAL.IS_ALARMS )
      I_Contact( "DB441_POWDER_FEEDERS_ALARM_DECODING".ALARMS_UNIT_01.POWDER_FEEDER[1].IS_ALARMS )
      I_Contact( "DB441_POWDER_FEEDERS_ALARM_DECODING".ALARMS_UNIT_02.POWDER_FEEDER[1].IS_ALARMS )
      I_Contact( "DB441_POWDER_FEEDERS_ALARM_DECODING".ALARMS_UNIT_02.POWDER_FEEDER[2].IS_ALARMS )
      Not()
      Coil( "DB441_POWDER_FEEDERS_ALARM_DECODING".GLOBAL_ALARMS_MACHINE.IS_ALARMS )
   END_RUNG
   // the same network as SCL:
   "DB441_POWDER_FEEDERS_ALARM_DECODING".GLOBAL_ALARMS_MACHINE.IS_ALARMS := NOT (NOT "DB441_POWDER_FEEDERS_ALARM_DECODING".ALARMS_CENTRAL.IS_ALARMS AND NOT "DB441_POWDER_FEEDERS_ALARM_DECODING".ALARMS_UNIT_01.POWDER_FEEDER[1].IS_ALARMS AND NOT "DB441_POWDER_FEEDERS_ALARM_DECODING".ALARMS_UNIT_02.POWDER_FEEDER[1].IS_ALARMS AND NOT "DB441_POWDER_FEEDERS_ALARM_DECODING".ALARMS_UNIT_02.POWDER_FEEDER[2].IS_ALARMS);
END_REGION

REGION Network 12: RETURN HOME POSITION ALARMS
   // Machine Emergency Return Alarm
   RUNG wire#powerrail
      I_Contact( "DB441_POWDER_FEEDERS_ALARM_DECODING".ALARMS_CENTRAL.RHP_ALARMS )
      I_Contact( "DB441_POWDER_FEEDERS_ALARM_DECODING".ALARMS_UNIT_01.POWDER_FEEDER[1].RHP_ALARMS )
      I_Contact( "DB441_POWDER_FEEDERS_ALARM_DECODING".ALARMS_UNIT_02.POWDER_FEEDER[1].RHP_ALARMS )
      I_Contact( "DB441_POWDER_FEEDERS_ALARM_DECODING".ALARMS_UNIT_02.POWDER_FEEDER[2].RHP_ALARMS )
      Not()
      Coil( "DB441_POWDER_FEEDERS_ALARM_DECODING".GLOBAL_ALARMS_MACHINE.RHP_ALARMS )
   END_RUNG
   // the same network as SCL:
   "DB441_POWDER_FEEDERS_ALARM_DECODING".GLOBAL_ALARMS_MACHINE.RHP_ALARMS := NOT (NOT "DB441_POWDER_FEEDERS_ALARM_DECODING".ALARMS_CENTRAL.RHP_ALARMS AND NOT "DB441_POWDER_FEEDERS_ALARM_DECODING".ALARMS_UNIT_01.POWDER_FEEDER[1].RHP_ALARMS AND NOT "DB441_POWDER_FEEDERS_ALARM_DECODING".ALARMS_UNIT_02.POWDER_FEEDER[1].RHP_ALARMS AND NOT "DB441_POWDER_FEEDERS_ALARM_DECODING".ALARMS_UNIT_02.POWDER_FEEDER[2].RHP_ALARMS);
END_REGION

REGION Network 13: STOP END OF CYCLE ALARMS
   // Machine End Of Cycle Alarm
   RUNG wire#powerrail
      I_Contact( "DB441_POWDER_FEEDERS_ALARM_DECODING".ALARMS_CENTRAL.SEOC_ALARMS )
      I_Contact( "DB441_POWDER_FEEDERS_ALARM_DECODING".ALARMS_UNIT_01.POWDER_FEEDER[1].SEOC_ALARMS )
      I_Contact( "DB441_POWDER_FEEDERS_ALARM_DECODING".ALARMS_UNIT_02.POWDER_FEEDER[1].SEOC_ALARMS )
      I_Contact( "DB441_POWDER_FEEDERS_ALARM_DECODING".ALARMS_UNIT_02.POWDER_FEEDER[2].SEOC_ALARMS )
      Not()
      Coil( "DB441_POWDER_FEEDERS_ALARM_DECODING".GLOBAL_ALARMS_MACHINE.SEOC_ALARMS )
   END_RUNG
   // the same network as SCL:
   "DB441_POWDER_FEEDERS_ALARM_DECODING".GLOBAL_ALARMS_MACHINE.SEOC_ALARMS := NOT (NOT "DB441_POWDER_FEEDERS_ALARM_DECODING".ALARMS_CENTRAL.SEOC_ALARMS AND NOT "DB441_POWDER_FEEDERS_ALARM_DECODING".ALARMS_UNIT_01.POWDER_FEEDER[1].SEOC_ALARMS AND NOT "DB441_POWDER_FEEDERS_ALARM_DECODING".ALARMS_UNIT_02.POWDER_FEEDER[1].SEOC_ALARMS AND NOT "DB441_POWDER_FEEDERS_ALARM_DECODING".ALARMS_UNIT_02.POWDER_FEEDER[2].SEOC_ALARMS);
END_REGION

REGION Network 14: IMMEDIATE STOP WARNING
   // Machine Full Stop Warning
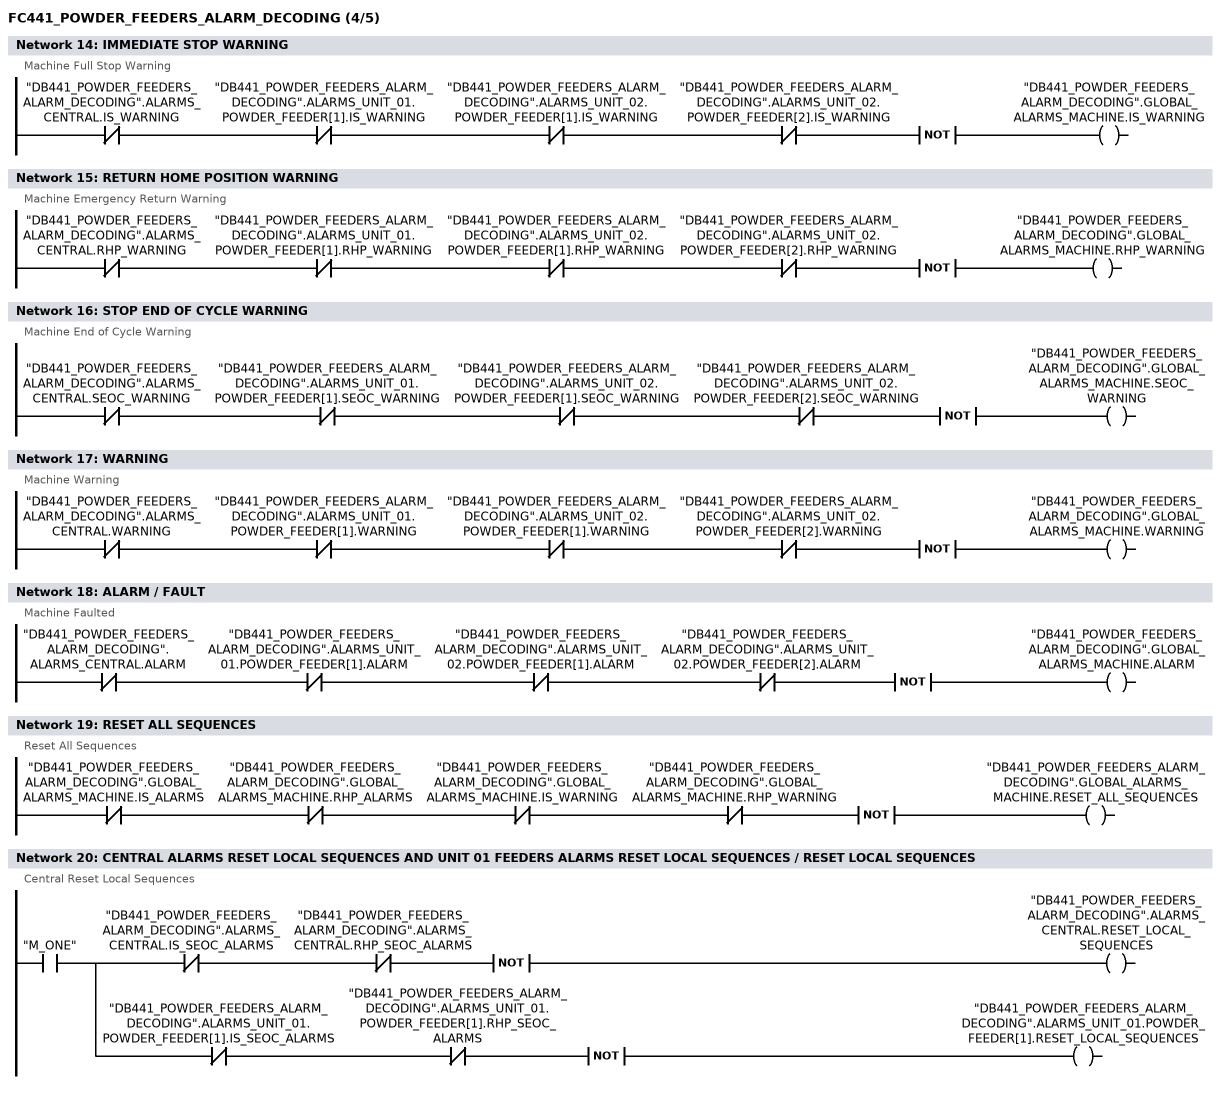
   RUNG wire#powerrail
      I_Contact( "DB441_POWDER_FEEDERS_ALARM_DECODING".ALARMS_CENTRAL.IS_WARNING )
      I_Contact( "DB441_POWDER_FEEDERS_ALARM_DECODING".ALARMS_UNIT_01.POWDER_FEEDER[1].IS_WARNING )
      I_Contact( "DB441_POWDER_FEEDERS_ALARM_DECODING".ALARMS_UNIT_02.POWDER_FEEDER[1].IS_WARNING )
      I_Contact( "DB441_POWDER_FEEDERS_ALARM_DECODING".ALARMS_UNIT_02.POWDER_FEEDER[2].IS_WARNING )
      Not()
      Coil( "DB441_POWDER_FEEDERS_ALARM_DECODING".GLOBAL_ALARMS_MACHINE.IS_WARNING )
   END_RUNG
   // the same network as SCL:
   "DB441_POWDER_FEEDERS_ALARM_DECODING".GLOBAL_ALARMS_MACHINE.IS_WARNING := NOT (NOT "DB441_POWDER_FEEDERS_ALARM_DECODING".ALARMS_CENTRAL.IS_WARNING AND NOT "DB441_POWDER_FEEDERS_ALARM_DECODING".ALARMS_UNIT_01.POWDER_FEEDER[1].IS_WARNING AND NOT "DB441_POWDER_FEEDERS_ALARM_DECODING".ALARMS_UNIT_02.POWDER_FEEDER[1].IS_WARNING AND NOT "DB441_POWDER_FEEDERS_ALARM_DECODING".ALARMS_UNIT_02.POWDER_FEEDER[2].IS_WARNING);
END_REGION

REGION Network 15: RETURN HOME POSITION WARNING
   // Machine Emergency Return Warning
   RUNG wire#powerrail
      I_Contact( "DB441_POWDER_FEEDERS_ALARM_DECODING".ALARMS_CENTRAL.RHP_WARNING )
      I_Contact( "DB441_POWDER_FEEDERS_ALARM_DECODING".ALARMS_UNIT_01.POWDER_FEEDER[1].RHP_WARNING )
      I_Contact( "DB441_POWDER_FEEDERS_ALARM_DECODING".ALARMS_UNIT_02.POWDER_FEEDER[1].RHP_WARNING )
      I_Contact( "DB441_POWDER_FEEDERS_ALARM_DECODING".ALARMS_UNIT_02.POWDER_FEEDER[2].RHP_WARNING )
      Not()
      Coil( "DB441_POWDER_FEEDERS_ALARM_DECODING".GLOBAL_ALARMS_MACHINE.RHP_WARNING )
   END_RUNG
   // the same network as SCL:
   "DB441_POWDER_FEEDERS_ALARM_DECODING".GLOBAL_ALARMS_MACHINE.RHP_WARNING := NOT (NOT "DB441_POWDER_FEEDERS_ALARM_DECODING".ALARMS_CENTRAL.RHP_WARNING AND NOT "DB441_POWDER_FEEDERS_ALARM_DECODING".ALARMS_UNIT_01.POWDER_FEEDER[1].RHP_WARNING AND NOT "DB441_POWDER_FEEDERS_ALARM_DECODING".ALARMS_UNIT_02.POWDER_FEEDER[1].RHP_WARNING AND NOT "DB441_POWDER_FEEDERS_ALARM_DECODING".ALARMS_UNIT_02.POWDER_FEEDER[2].RHP_WARNING);
END_REGION

REGION Network 16: STOP END OF CYCLE WARNING
   // Machine End of Cycle Warning
   RUNG wire#powerrail
      I_Contact( "DB441_POWDER_FEEDERS_ALARM_DECODING".ALARMS_CENTRAL.SEOC_WARNING )
      I_Contact( "DB441_POWDER_FEEDERS_ALARM_DECODING".ALARMS_UNIT_01.POWDER_FEEDER[1].SEOC_WARNING )
      I_Contact( "DB441_POWDER_FEEDERS_ALARM_DECODING".ALARMS_UNIT_02.POWDER_FEEDER[1].SEOC_WARNING )
      I_Contact( "DB441_POWDER_FEEDERS_ALARM_DECODING".ALARMS_UNIT_02.POWDER_FEEDER[2].SEOC_WARNING )
      Not()
      Coil( "DB441_POWDER_FEEDERS_ALARM_DECODING".GLOBAL_ALARMS_MACHINE.SEOC_WARNING )
   END_RUNG
   // the same network as SCL:
   "DB441_POWDER_FEEDERS_ALARM_DECODING".GLOBAL_ALARMS_MACHINE.SEOC_WARNING := NOT (NOT "DB441_POWDER_FEEDERS_ALARM_DECODING".ALARMS_CENTRAL.SEOC_WARNING AND NOT "DB441_POWDER_FEEDERS_ALARM_DECODING".ALARMS_UNIT_01.POWDER_FEEDER[1].SEOC_WARNING AND NOT "DB441_POWDER_FEEDERS_ALARM_DECODING".ALARMS_UNIT_02.POWDER_FEEDER[1].SEOC_WARNING AND NOT "DB441_POWDER_FEEDERS_ALARM_DECODING".ALARMS_UNIT_02.POWDER_FEEDER[2].SEOC_WARNING);
END_REGION

REGION Network 17: WARNING
   // Machine Warning
   RUNG wire#powerrail
      I_Contact( "DB441_POWDER_FEEDERS_ALARM_DECODING".ALARMS_CENTRAL.WARNING )
      I_Contact( "DB441_POWDER_FEEDERS_ALARM_DECODING".ALARMS_UNIT_01.POWDER_FEEDER[1].WARNING )
      I_Contact( "DB441_POWDER_FEEDERS_ALARM_DECODING".ALARMS_UNIT_02.POWDER_FEEDER[1].WARNING )
      I_Contact( "DB441_POWDER_FEEDERS_ALARM_DECODING".ALARMS_UNIT_02.POWDER_FEEDER[2].WARNING )
      Not()
      Coil( "DB441_POWDER_FEEDERS_ALARM_DECODING".GLOBAL_ALARMS_MACHINE.WARNING )
   END_RUNG
   // the same network as SCL:
   "DB441_POWDER_FEEDERS_ALARM_DECODING".GLOBAL_ALARMS_MACHINE.WARNING := NOT (NOT "DB441_POWDER_FEEDERS_ALARM_DECODING".ALARMS_CENTRAL.WARNING AND NOT "DB441_POWDER_FEEDERS_ALARM_DECODING".ALARMS_UNIT_01.POWDER_FEEDER[1].WARNING AND NOT "DB441_POWDER_FEEDERS_ALARM_DECODING".ALARMS_UNIT_02.POWDER_FEEDER[1].WARNING AND NOT "DB441_POWDER_FEEDERS_ALARM_DECODING".ALARMS_UNIT_02.POWDER_FEEDER[2].WARNING);
END_REGION

REGION Network 18: ALARM / FAULT
   // Machine Faulted
   RUNG wire#powerrail
      I_Contact( "DB441_POWDER_FEEDERS_ALARM_DECODING".ALARMS_CENTRAL.ALARM )
      I_Contact( "DB441_POWDER_FEEDERS_ALARM_DECODING".ALARMS_UNIT_01.POWDER_FEEDER[1].ALARM )
      I_Contact( "DB441_POWDER_FEEDERS_ALARM_DECODING".ALARMS_UNIT_02.POWDER_FEEDER[1].ALARM )
      I_Contact( "DB441_POWDER_FEEDERS_ALARM_DECODING".ALARMS_UNIT_02.POWDER_FEEDER[2].ALARM )
      Not()
      Coil( "DB441_POWDER_FEEDERS_ALARM_DECODING".GLOBAL_ALARMS_MACHINE.ALARM )
   END_RUNG
   // the same network as SCL:
   "DB441_POWDER_FEEDERS_ALARM_DECODING".GLOBAL_ALARMS_MACHINE.ALARM := NOT (NOT "DB441_POWDER_FEEDERS_ALARM_DECODING".ALARMS_CENTRAL.ALARM AND NOT "DB441_POWDER_FEEDERS_ALARM_DECODING".ALARMS_UNIT_01.POWDER_FEEDER[1].ALARM AND NOT "DB441_POWDER_FEEDERS_ALARM_DECODING".ALARMS_UNIT_02.POWDER_FEEDER[1].ALARM AND NOT "DB441_POWDER_FEEDERS_ALARM_DECODING".ALARMS_UNIT_02.POWDER_FEEDER[2].ALARM);
END_REGION

REGION Network 19: RESET ALL SEQUENCES
   // Reset All Sequences
   RUNG wire#powerrail
      I_Contact( "DB441_POWDER_FEEDERS_ALARM_DECODING".GLOBAL_ALARMS_MACHINE.IS_ALARMS )
      I_Contact( "DB441_POWDER_FEEDERS_ALARM_DECODING".GLOBAL_ALARMS_MACHINE.RHP_ALARMS )
      I_Contact( "DB441_POWDER_FEEDERS_ALARM_DECODING".GLOBAL_ALARMS_MACHINE.IS_WARNING )
      I_Contact( "DB441_POWDER_FEEDERS_ALARM_DECODING".GLOBAL_ALARMS_MACHINE.RHP_WARNING )
      Not()
      Coil( "DB441_POWDER_FEEDERS_ALARM_DECODING".GLOBAL_ALARMS_MACHINE.RESET_ALL_SEQUENCES )
   END_RUNG
   // the same network as SCL:
   "DB441_POWDER_FEEDERS_ALARM_DECODING".GLOBAL_ALARMS_MACHINE.RESET_ALL_SEQUENCES := NOT (NOT "DB441_POWDER_FEEDERS_ALARM_DECODING".GLOBAL_ALARMS_MACHINE.IS_ALARMS AND NOT "DB441_POWDER_FEEDERS_ALARM_DECODING".GLOBAL_ALARMS_MACHINE.RHP_ALARMS AND NOT "DB441_POWDER_FEEDERS_ALARM_DECODING".GLOBAL_ALARMS_MACHINE.IS_WARNING AND NOT "DB441_POWDER_FEEDERS_ALARM_DECODING".GLOBAL_ALARMS_MACHINE.RHP_WARNING);
END_REGION

REGION Network 20: CENTRAL ALARMS RESET LOCAL SEQUENCES AND UNIT 01 FEEDERS ALARMS RESET LOCAL SEQUENCES / RESET LOCAL SEQUENCES
   // Central Reset Local Sequences
   RUNG wire#powerrail
      Contact( "M_ONE" )
      wire#w1
      I_Contact( "DB441_POWDER_FEEDERS_ALARM_DECODING".ALARMS_CENTRAL.IS_SEOC_ALARMS )
      I_Contact( "DB441_POWDER_FEEDERS_ALARM_DECODING".ALARMS_CENTRAL.RHP_SEOC_ALARMS )
      Not()
      Coil( "DB441_POWDER_FEEDERS_ALARM_DECODING".ALARMS_CENTRAL.RESET_LOCAL_SEQUENCES )
   END_RUNG
   RUNG wire#w1
      I_Contact( "DB441_POWDER_FEEDERS_ALARM_DECODING".ALARMS_UNIT_01.POWDER_FEEDER[1].IS_SEOC_ALARMS )
      I_Contact( "DB441_POWDER_FEEDERS_ALARM_DECODING".ALARMS_UNIT_01.POWDER_FEEDER[1].RHP_SEOC_ALARMS )
      Not()
      Coil( "DB441_POWDER_FEEDERS_ALARM_DECODING".ALARMS_UNIT_01.POWDER_FEEDER[1].RESET_LOCAL_SEQUENCES )
   END_RUNG
   // the same network as SCL:
   "DB441_POWDER_FEEDERS_ALARM_DECODING".ALARMS_CENTRAL.RESET_LOCAL_SEQUENCES := NOT ("M_ONE" AND NOT "DB441_POWDER_FEEDERS_ALARM_DECODING".ALARMS_CENTRAL.IS_SEOC_ALARMS AND NOT "DB441_POWDER_FEEDERS_ALARM_DECODING".ALARMS_CENTRAL.RHP_SEOC_ALARMS);
   "DB441_POWDER_FEEDERS_ALARM_DECODING".ALARMS_UNIT_01.POWDER_FEEDER[1].RESET_LOCAL_SEQUENCES := NOT ("M_ONE" AND NOT "DB441_POWDER_FEEDERS_ALARM_DECODING".ALARMS_UNIT_01.POWDER_FEEDER[1].IS_SEOC_ALARMS AND NOT "DB441_POWDER_FEEDERS_ALARM_DECODING".ALARMS_UNIT_01.POWDER_FEEDER[1].RHP_SEOC_ALARMS);
END_REGION

REGION Network 21: UNIT 02 FEEDERS ALARMS RESET LOCAL SEQUENCES / RESET LOCAL SEQUENCES
   // Central Reset Local Sequences
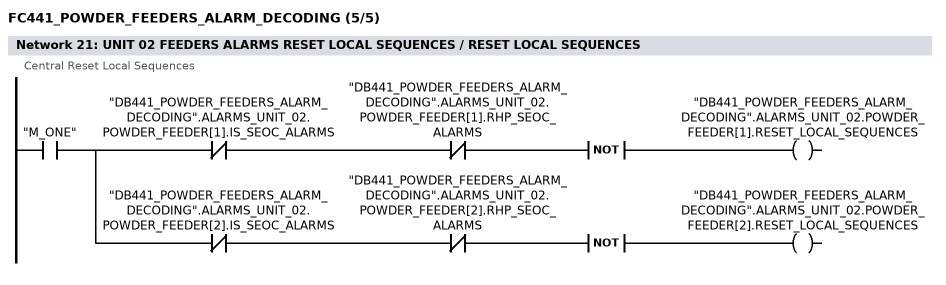
   RUNG wire#powerrail
      Contact( "M_ONE" )
      wire#w1
      I_Contact( "DB441_POWDER_FEEDERS_ALARM_DECODING".ALARMS_UNIT_02.POWDER_FEEDER[1].IS_SEOC_ALARMS )
      I_Contact( "DB441_POWDER_FEEDERS_ALARM_DECODING".ALARMS_UNIT_02.POWDER_FEEDER[1].RHP_SEOC_ALARMS )
      Not()
      Coil( "DB441_POWDER_FEEDERS_ALARM_DECODING".ALARMS_UNIT_02.POWDER_FEEDER[1].RESET_LOCAL_SEQUENCES )
   END_RUNG
   RUNG wire#w1
      I_Contact( "DB441_POWDER_FEEDERS_ALARM_DECODING".ALARMS_UNIT_02.POWDER_FEEDER[2].IS_SEOC_ALARMS )
      I_Contact( "DB441_POWDER_FEEDERS_ALARM_DECODING".ALARMS_UNIT_02.POWDER_FEEDER[2].RHP_SEOC_ALARMS )
      Not()
      Coil( "DB441_POWDER_FEEDERS_ALARM_DECODING".ALARMS_UNIT_02.POWDER_FEEDER[2].RESET_LOCAL_SEQUENCES )
   END_RUNG
   // the same network as SCL:
   "DB441_POWDER_FEEDERS_ALARM_DECODING".ALARMS_UNIT_02.POWDER_FEEDER[1].RESET_LOCAL_SEQUENCES := NOT ("M_ONE" AND NOT "DB441_POWDER_FEEDERS_ALARM_DECODING".ALARMS_UNIT_02.POWDER_FEEDER[1].IS_SEOC_ALARMS AND NOT "DB441_POWDER_FEEDERS_ALARM_DECODING".ALARMS_UNIT_02.POWDER_FEEDER[1].RHP_SEOC_ALARMS);
   "DB441_POWDER_FEEDERS_ALARM_DECODING".ALARMS_UNIT_02.POWDER_FEEDER[2].RESET_LOCAL_SEQUENCES := NOT ("M_ONE" AND NOT "DB441_POWDER_FEEDERS_ALARM_DECODING".ALARMS_UNIT_02.POWDER_FEEDER[2].IS_SEOC_ALARMS AND NOT "DB441_POWDER_FEEDERS_ALARM_DECODING".ALARMS_UNIT_02.POWDER_FEEDER[2].RHP_SEOC_ALARMS);
END_REGION
END_FUNCTION
